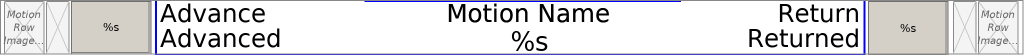
VISUALIZATION ModeRow  // 1024x55
VAR_IN_OUT
	MotionRowInstanceSingle:typeMotionRow; //feedback to motion row to operator
	MotionRowButtonsSingle:typeMotionRowButtons; //button feedback in seperate interface
END_VAR
    Rectangle (155,0 710x55), invisible if: MotionRowInstanceSingle.Returned.bHideCoil AND MotionRowInstanceSingle.bHideName
    Button (868,1 80x55), "%s", text variable: MotionRowInstanceSingle.Returned.NumberOrder, invisible if: MotionRowInstanceSingle.Returned.bHideButton
        tap MotionRowButtonsSingle.btnReturn
    Button (71,1 80x53), "%s", text variable: MotionRowInstanceSingle.Advance.NumberOrder, invisible if: MotionRowInstanceSingle.Advance.bHideButton
        tap MotionRowButtonsSingle.btnAdvance
    Rectangle (393,25 273x33), "%s", text variable: MotionRowInstanceSingle.strPosn, invisible if: MotionRowInstanceSingle.bHidePosn
    Group (157,1 706x52)
        Rectangle (524,0 182x25), "Return", invisible if: MotionRowInstanceSingle.Returned.bHideCoil or MotionRowInstanceSingle.bIsAbsSymSwitch, text list: 'ModeRowText', text index: MotionRowInstanceSingle.IndexLocation + 3, colour variable: MotionRowInstanceSingle.Returned.CoilColour
        Rectangle (235,0 273x25), "Motion Name", invisible if: MotionRowInstanceSingle.bHideName or MotionRowInstanceSingle.bIsAbsSymSwitch, text list: 'ModeRowText', text index: MotionRowInstanceSingle.IndexLocation + 6
        Rectangle (524,25 182x25), "Returned", invisible if: MotionRowInstanceSingle.Returned.bHideDepth or MotionRowInstanceSingle.bIsAbsSymSwitch, text list: 'ModeRowText', text index: MotionRowInstanceSingle.IndexLocation + 4, colour variable: MotionRowInstanceSingle.Returned.FdbkColour
        Rectangle (0,0 207x25), "Advance", text variable: MotionRowInstanceSingle.Advance.valCoil, invisible if: MotionRowInstanceSingle.Advance.bHideCoil or MotionRowInstanceSingle.bIsAbsSymSwitch, text list: 'ModeRowText', text index: MotionRowInstanceSingle.IndexLocation + 0, colour variable: MotionRowInstanceSingle.Advance.CoilColour
        Rectangle (0,25 207x25), "Advanced", invisible if: MotionRowInstanceSingle.Advance.bHideDepth or MotionRowInstanceSingle.bIsAbsSymSwitch, text list: 'ModeRowText', text index: MotionRowInstanceSingle.IndexLocation + 1, colour variable: MotionRowInstanceSingle.Advance.FdbkColour
    Image (4,1 40x53), invisible if: NOT MotionRowInstanceSingle.Advance.InterlockOK OR MotionRowInstanceSingle.Advance.bHideInterlock, image: MotionRowImages.LeftHighlight
    Image (4,1 40x53), invisible if: MotionRowInstanceSingle.Advance.InterlockOK OR MotionRowInstanceSingle.Advance.bHideInterlock, image: MotionRowImages.LeftNot
    Image (978,1 40x53), invisible if: MotionRowInstanceSingle.Returned.InterlockOK OR MotionRowInstanceSingle.Returned.bHideInterlock, image: MotionRowImages.RightNot
    Image (978,1 40x53), invisible if: NOT MotionRowInstanceSingle.Returned.InterlockOK OR MotionRowInstanceSingle.Returned.bHideInterlock, image: MotionRowImages.RightHighlight
    Image (46,1 23x53), invisible if: MotionRowInstanceSingle.Advance.Prompt OR MotionRowInstanceSingle.Advance.bHidePrompt, image: MotionRowImages.PromptNOK
    Image (953,1 23x53), invisible if: NOT MotionRowInstanceSingle.Returned.Prompt OR MotionRowInstanceSingle.Returned.bHidePrompt, image: MotionRowImages.PromptOK
    Image (953,1 23x53), invisible if: MotionRowInstanceSingle.Returned.Prompt OR MotionRowInstanceSingle.Returned.bHidePrompt, image: MotionRowImages.PromptNOK
    Image (46,1 23x53), invisible if: NOT MotionRowInstanceSingle.Advance.Prompt OR MotionRowInstanceSingle.Advance.bHidePrompt, image: MotionRowImages.PromptOK
    Group (157,1 706x52)
        Rectangle (524,0 182x25), "Return", invisible if: MotionRowInstanceSingle.Returned.bHideCoil or NOT MotionRowInstanceSingle.bIsAbsSymSwitch, text list: 'ModeRowText', text index: MotionRowInstanceSingle.IndexLocation + 3 + 10, colour variable: MotionRowInstanceSingle.Returned.CoilColour
        Rectangle (235,0 273x25), "Motion Name", invisible if: MotionRowInstanceSingle.bHideName or NOT MotionRowInstanceSingle.bIsAbsSymSwitch, text list: 'ModeRowText', text index: MotionRowInstanceSingle.IndexLocation + 6 + 10
        Rectangle (524,25 182x25), "Returned", invisible if: MotionRowInstanceSingle.Returned.bHideDepth or NOT MotionRowInstanceSingle.bIsAbsSymSwitch, text list: 'ModeRowText', text index: MotionRowInstanceSingle.IndexLocation + 4 + 10, colour variable: MotionRowInstanceSingle.Returned.FdbkColour
        Rectangle (0,0 207x25), "Advance", text variable: MotionRowInstanceSingle.Advance.valCoil, invisible if: MotionRowInstanceSingle.Advance.bHideCoil or NOT MotionRowInstanceSingle.bIsAbsSymSwitch, text list: 'ModeRowText', text index: MotionRowInstanceSingle.IndexLocation + 0 + 10, colour variable: MotionRowInstanceSingle.Advance.CoilColour
        Rectangle (0,25 207x25), "Advanced", invisible if: MotionRowInstanceSingle.Advance.bHideDepth or NOT MotionRowInstanceSingle.bIsAbsSymSwitch, text list: 'ModeRowText', text index: MotionRowInstanceSingle.IndexLocation + 1 + 10, colour variable: MotionRowInstanceSingle.Advance.FdbkColour
END_VISUALIZATION

(* stored: Version 1.1.0.1, ProductVersion 3.1.4024.12
   Visu ModeRow: Id {e90b3459-e2be-49ef-90ff-65a7d8343fc1} *)
